# EPICS substitutions: hmp40x0/Db/hmp40x0.substitutions
file "hmp40x0-gen.template" { pattern
{}
{}
}

file "hmp40x0-chan.template" { pattern
{CHAN}
{1}
{2}
{3}
{4}
}
